{attribute 'OPC.UA.DA' := '1'}
FUNCTION_BLOCK PhotoLumChamber EXTENDS ChamberBase
VAR_INPUT
	IoChamberPhotoLum : IoChamberPhotoLum;
END_VAR
VAR_OUTPUT
END_VAR
VAR
	{attribute 'OPC.UA.DA' := '0'}
	_config : PhotoLumChamberConfig;	
	
	{attribute 'OPC.UA.DA' := '0'}
	_initDevice : BOOL;
	
	{attribute 'OPC.UA.DA' := '0'}
	_itemInit : INT;
	{attribute 'OPC.UA.DA' := '0'}
	_itemScheduler : INT;
	{attribute 'OPC.UA.DA' := '0'}
	_itemExecScheduler : INT;		
	{attribute 'OPC.UA.DA' := '0'}
	_itemRaisedProperties : INT;			
	{attribute 'OPC.UA.DA' := '0'}
	_pulseGenerator : TON;	
	
	{region 'Commands'}	
		 	
	{attribute 'OPC.UA.DA' := '0'}
	_enableCamera : BOOL;
	{attribute 'OPC.UA.DA' := '0'}
	_moveSlitDoorPositionCmd	 : BOOL;	
	{attribute 'OPC.UA.DA' := '0'}			  		   
	_raisePropertiesCmd : BOOL;	 
			
	{endregion}
	
	{attribute 'OPC.UA.DA' := '0'}
	_deliverMessages : INT;
	
	InterlockPanelsMsg : STRING(255);
	SlitDoorPositionMsg : STRING(255);
	SlitDoorOpenPositionMsg : STRING(255);
	SlitDoorClosePositionMsg : STRING(255);
	
	{attribute 'OPC.UA.DA' := '0'}
	message : STRING(255);
	
	{attribute 'OPC.UA.DA' := '0'}
	_pos : INT;	
	
	{attribute 'OPC.UA.DA' := '0'}
	tmpConcat1 : STRING;
	{attribute 'OPC.UA.DA' := '0'}
	tmpConcat2 : STRING;
	{attribute 'OPC.UA.DA' := '0'}
	tmpConcatName : STRING; 
	{attribute 'OPC.UA.DA' := '0'}
	tmpConcatDescription : STRING;
	{attribute 'OPC.UA.DA' := '0'}
	tmpConcatInterlockID : STRING;
	
	{attribute 'OPC.UA.DA' := '0'}
	_itemInterlock : UINT;
	{attribute 'OPC.UA.DA' := '0'}
	_interlockCount : UINT;			
END_VAR

SUPER^();

// Init device
InitDevice(); 

// Deliver messages
CASE _deliverMessages OF	
	EFeedbackMsgPhotoLumChamber.InterlockPanelsMsg :
		InterlockPanelsMsg := message;	
	EFeedbackMsgPhotoLumChamber.SlitDoorPositionMsg :
		SlitDoorPositionMsg := TO_STRING(SlitDoorPosition);		
	EFeedbackMsgPhotoLumChamber.SlitDoorOpenPositionMsg :
		SlitDoorOpenPositionMsg := TO_STRING(SlitDoorOpenPosition);	
	EFeedbackMsgPhotoLumChamber.SlitDoorClosePositionMsg :
		SlitDoorClosePositionMsg := TO_STRING(SlitDoorClosePosition);		
END_CASE

// Commands
MoveSlitDoorPosition(_moveSlitDoorPositionCmd, _pos); 
RaisePropertiesChanged(_raisePropertiesCmd);

IF NOT _moveSlitDoorPositionCmd AND NOT _raisePropertiesCmd THEN	
	MessageScheduler();
END_IF

METHOD FB_init : BOOL
VAR_INPUT
	bInitRetains : BOOL; // if TRUE, the retain variables are initialized (warm start / cold start)
	bInCopyCode : BOOL;  // if TRUE, the instance afterwards gets moved into the copy code (online change)
	Config : PhotoLumChamberConfig;
END_VAR
IF Config.IsEnabled THEN
	_config := Config;	

	SUPER^._chamberConfig.Name := Config.Name;
	SUPER^._chamberConfig.DeviceID := Config.DeviceID;
	SUPER^._chamberConfig.IsEnabled := Config.IsEnabled;
	SUPER^._chamberConfig.LogLevel := Config.LogLevel;
	
	SUPER^.Name := Config.Name;
	SUPER^.DeviceID := Config.DeviceID;
	
	THIS^.Family := DeviceFamily.Chamber;

	THIS^.SetReady();
	_Logger.Information(_message.Reset().Append('Init ').
							Append('{').Append(TO_STRING(THIS^.Family)).Append('} - ').
							Append('{').Append(TO_STRING(THIS^.Name)).Append('} - ').
							Append('Status : ').Append(TO_STRING(THIS^.Status)).
							ToString());										 
END_IF
END_METHOD

METHOD InitDevice
VAR_INPUT
END_VAR
IF NOT _initDevice THEN			
	_logger.Information(_message.Reset().
								Append(_config.Name).
								Append(' - init device').ToString());		
							
	_initDevice := TRUE;
	
END_IF
END_METHOD

METHOD MessageScheduler
VAR_INPUT
END_VAR
IF _pulseGenerator.Q THEN
	_pulseGenerator(IN := FALSE, PT := T#10MS);
		
	CASE _itemScheduler OF	
		0: SlitDoorPositionMsg := ' ';
		   _itemScheduler := 1;
		   
		1: ReadInterlock();
		   _itemScheduler := 2;
	
		2:  ReadSlitDoorPosition();
			_itemScheduler := 3;

		3:  ReadSlitDoorOpenPosition();
			_itemScheduler := 4;

		4:  ReadSlitDoorClosePosition();
			_itemScheduler := 0;					
	END_CASE
ELSE
	_pulseGenerator(IN := TRUE, PT := T#50MS);		
END_IF
END_METHOD

{attribute 'TcRpcEnable' := '1'}
METHOD MoveSlitDoorPosition
VAR_INPUT
	Execute : BOOL;
	Position : INT;
END_VAR
IF Execute THEN
	_logger.Information(_message.Reset().Append(_config.Name).Append(' - Move slit door position : ').Append(TO_STRING(Position)).ToString());
	
	_moveSlitDoorPositionCmd := FALSE;
		
	IF Position = ESlitDoorPosition.Open THEN
		IoChamberPhotoLum.OutputOpenSlitDoor := TRUE;
		IoChamberPhotoLum.OutputCloseSlitDoor := FALSE;
	ELSIF Position = ESlitDoorPosition.Close THEN
		IoChamberPhotoLum.OutputOpenSlitDoor := FALSE;
		IoChamberPhotoLum.OutputCloseSlitDoor := TRUE;
		
		//IsInLoadingPosition := FALSE;
	ELSE
		_logger.Error(_message.Reset().Append(_config.Name).Append(' - unknown position : ').Append(TO_STRING(Position)).ToString());
		
		//IsInLoadingPosition := FALSE;
	END_IF
				
	_itemScheduler := 0;
END_IF
END_METHOD

{attribute 'TcRpcEnable' := '1'}
METHOD RaisePropertiesChanged
VAR_INPUT
	Execute : BOOL;
END_VAR
IF Execute THEN		
	_raisePropertiesCmd := TRUE;	
		
	IF _pulseGenerator.Q THEN
		_pulseGenerator(IN := FALSE, PT := T#10MS);
		
		CASE _itemRaisedProperties OF		
			0: 	SUPER^._raisePropertiesBase := TRUE;		   
				_itemRaisedProperties := 10;
				
			10: _logger.Information(_message.Reset().Append(_config.Name).Append(' - RaisePropertiesChanged').ToString());
				_raisePropertiesCmd := FALSE;
				_itemRaisedProperties := 0;
		END_CASE	
	ELSE
		_pulseGenerator(IN := TRUE, PT := T#50MS);	
	END_IF		
END_IF
END_METHOD

METHOD ReadInterlock 
VAR_INPUT
END_VAR
VAR
	statePanel : STRING;
END_VAR
_deliverMessages := EFeedbackMsgPsdChamber.InterlockPanelsMsg;

IF _interlockCount < Const.PHOTOLUM_NUMBER_INTERLOCK_PANELS - 1 THEN
	_interlockCount := _interlockCount + 1;
ELSE
	_interlockCount := 0;
END_IF

tmpConcatName := CONCAT(_config.Interlock[_interlockCount].Name, ';');
tmpConcatDescription := CONCAT(_config.Interlock[_interlockCount].Description, ';');
tmpConcatInterlockID := CONCAT(UINT_TO_STRING(_config.Interlock[_interlockCount].InterlockID), ';');

tmpConcat1 := CONCAT(tmpConcatName, tmpConcatDescription);
tmpConcat2 := CONCAT(tmpConcat1, tmpConcatInterlockID);

IF _config.Interlock[_interlockCount].State THEN
	statePanel := 'Closed';
ELSE
	statePanel := 'Opened';
END_IF

message := CONCAT(tmpConcat2, statePanel);
END_METHOD

METHOD ReadSlitDoorClosePosition
VAR_INPUT
END_VAR
VAR
	open : BOOL;
	close : BOOL;
END_VAR
_deliverMessages := EFeedbackMsgPhotoLumChamber.SlitDoorClosePositionMsg;
SlitDoorClosePosition := IoChamberPhotoLum.InputCloseSlitDoor;
END_METHOD

METHOD ReadSlitDoorOpenPosition
VAR_INPUT
END_VAR
_deliverMessages := EFeedbackMsgPhotoLumChamber.SlitDoorOpenPositionMsg;
SlitDoorOpenPosition := IoChamberPhotoLum.InputOpenSlitDoor;
END_METHOD

METHOD ReadSlitDoorPosition
VAR_INPUT
END_VAR
VAR
	open : BOOL;
	close : BOOL;
END_VAR
_deliverMessages := EFeedbackMsgPhotoLumChamber.SlitDoorPositionMsg;

open := IoChamberPhotoLum.InputOpenSlitDoor;
close := IoChamberPhotoLum.InputCloseSlitDoor;

IF open AND NOT close THEN
	IoChamberPhotoLum.EfemInterlockSlitDoor := TRUE;	
	IoChamberPhotoLum.EfemInterlockArmExtendedEnable := TRUE;	
	SlitDoorPosition := ESlitDoorPosition.Open;	
ELSIF close AND NOT open THEN
	IoChamberPhotoLum.EfemInterlockSlitDoor := FALSE;
	IoChamberPhotoLum.EfemInterlockArmExtendedEnable := FALSE;
	SlitDoorPosition := ESlitDoorPosition.Close;
ELSIF close AND open THEN
	IoChamberPhotoLum.EfemInterlockSlitDoor := FALSE;
	IoChamberPhotoLum.EfemInterlockArmExtendedEnable := FALSE;
	SlitDoorPosition := ESlitDoorPosition.Error;	
ELSE
	IoChamberPhotoLum.EfemInterlockSlitDoor := FALSE;
	IoChamberPhotoLum.EfemInterlockArmExtendedEnable := FALSE;
	SlitDoorPosition := ESlitDoorPosition.Unknown;		
END_IF
END_METHOD

END_FUNCTION_BLOCK

(* stored: Version 1.1.0.1, ProductVersion 3.1.4024.12
   POU PhotoLumChamber: Id {50f08ae1-454c-45a7-9405-3d74b783e25e}, SpecialFunc None
   Folder Commands: Id {98986a00-5521-4856-953b-50097e90aa42}
   Method FB_init: Id {07ddbfcf-e42d-47c0-b42a-69d4f2f4abee}
   Method InitDevice: Id {47ccf362-cff8-4605-b81d-bdf4b6fe9599}
   Method MessageScheduler: Id {f40e75a0-b5f6-4cd1-99da-a1cd39ddcdc6}
   Method MoveSlitDoorPosition: Id {2adb4c20-3cad-4872-8478-a1e267ea3098}
   Method RaisePropertiesChanged: Id {daf67c55-7929-45d5-b907-80dc69801af5}
   Method ReadInterlock: Id {11398588-9f18-4476-a7dd-e69fe8066d70}
   Method ReadSlitDoorClosePosition: Id {b3f9a4a8-9a30-4200-8666-50f17637f3b4}
   Method ReadSlitDoorOpenPosition: Id {94d18b75-d3bc-4952-a8a4-b30cbadf5c64}
   Method ReadSlitDoorPosition: Id {8e56b65e-fe0b-49c8-ae52-ad1e8ef617f2} *)
